// TwinCAT 3 PLC project PLC_SerialCom_Sample1
// ProgramVersion: 3.1.0.8
// libraries:
//   Tc2_SerialCom, * (Beckhoff Automation GmbH)
//   Tc2_Standard, * (Beckhoff Automation GmbH)
//   Tc3_Module, * (Beckhoff Automation GmbH)
// project tree:
//   GVLs/ GVL.TcGVL (not stored)
//   / PlcTask_Fast.TcTTO (not stored), PlcTask_Standard.TcTTO (not stored)
//   POUs/ Background.TcPOU (not stored), BackgroundEL.TcPOU (not stored), FB_Receive.TcPOU, FB_Send.TcPOU (not stored), FB_SerialCom.TcPOU (not stored), MAIN.TcPOU (not stored)

// ---- POUs/FB_Receive.TcPOU
FUNCTION_BLOCK FB_Receive
VAR_IN_OUT
	TxBuffer	: ComBuffer;
	RxBuffer	: ComBuffer;
END_VAR
VAR
	//Timer		: TON := (PT:=T#1S);
	//fbSend		: SendString;
	//bSendBusy	: BOOL;
	//eSendErrorID: ComError_t;
	//bReceivedByte	: BYTE;
	//bByteReceived	: BOOL;
	//bReceiveBusy	: BOOL;
	//bReceiveError	: BOOL;
	//bReceiveTimeout	: BOOL;
	fbReceive		: ReceiveByte;
	nReceiveCounter	: UDINT;
	bLastReceivedByte: BYTE;
	eReceiveErrorID	: ComError_t;
END_VAR

fbReceive(
//	Prefix:= '$02',
//	Suffix:= '$03',
//	Timeout:= T#1s,
//	ReceivedString:= bReceivedByte,
//	RxTimeout=> bReceiveTimeout 
//	ByteReceived=> bByteReceived,
//	Busy=> bReceiveBusy,
	RXbuffer:= RxBuffer,
	Error=> ,
	ByteReceived=>,
	ReceivedByte=>,
	);
IF fbReceive.Error <> COMERROR_NOERROR THEN
	eReceiveErrorID := fbReceive.Error;
END_IF
IF fbReceive.ByteReceived THEN
	nReceiveCounter := nReceiveCounter + 1;
	bLastReceivedByte := fbReceive.ReceivedByte;
END_IF

END_FUNCTION_BLOCK
